{attribute 'GeneratedUsingTerminal: EL1262-0000-0002'}
{attribute addProperty BoxType "EL1262-0000-0002"}
{attribute addProperty Id "EtcSlaveTerminalBaseCh1_CycleCountAT %I*Ch1_CycleCount_9DBE2BC52Ch1_Input_0AT %I*Ch1_Input_FFC4CE241Ch1_Input_1AT %I*Ch1_Input_FFC4CE241Ch1_Input_2AT %I*Ch1_Input_FFC4CE241Ch1_Input_3AT %I*Ch1_Input_FFC4CE241Ch1_Input_4AT %I*Ch1_Input_FFC4CE241Ch1_Input_5AT %I*Ch1_Input_FFC4CE241Ch1_Input_6AT %I*Ch1_Input_FFC4CE241Ch1_Input_7AT %I*Ch1_Input_FFC4CE241Ch1_Input_8AT %I*Ch1_Input_FFC4CE241Ch1_Input_9AT %I*Ch1_Input_FFC4CE241GapAT %I*EMPTY_STRUCTURE0Ch2_CycleCountAT %I*Ch2_CycleCount_976A51B52Ch2_Input_0AT %I*Ch2_Input_78ADA90C1Ch2_Input_1AT %I*Ch2_Input_78ADA90C1Ch2_Input_2AT %I*Ch2_Input_78ADA90C1Ch2_Input_3AT %I*Ch2_Input_78ADA90C1Ch2_Input_4AT %I*Ch2_Input_78ADA90C1Ch2_Input_5AT %I*Ch2_Input_78ADA90C1Ch2_Input_6AT %I*Ch2_Input_78ADA90C1Ch2_Input_7AT %I*Ch2_Input_78ADA90C1Ch2_Input_8AT %I*Ch2_Input_78ADA90C1Ch2_Input_9AT %I*Ch2_Input_78ADA90C1Gap_1AT %I*EMPTY_STRUCTURE0NextSync1TimeAT %I*NextSync1Time_EE185E174WcStateAT %I*WcState_9091E0EB2InfoDataAT %I*InfoData_A7436BC610"}
{attribute addProperty CRC "3126613733"}
{attribute addProperty Size "40"}
TYPE EL1262_BA5C56E5 EXTENDS EtcSlaveTerminalBase :
STRUCT
	{attribute addProperty Name "Ch1_CycleCount"}
	Ch1_CycleCount : Ch1_CycleCount_9DBE2BC5;
	{attribute addProperty Name "Ch1_Input_0"}
	Ch1_Input_0 : Ch1_Input_FFC4CE24;
	{attribute addProperty Name "Ch1_Input_1"}
	Ch1_Input_1 : Ch1_Input_FFC4CE24;
	{attribute addProperty Name "Ch1_Input_2"}
	Ch1_Input_2 : Ch1_Input_FFC4CE24;
	{attribute addProperty Name "Ch1_Input_3"}
	Ch1_Input_3 : Ch1_Input_FFC4CE24;
	{attribute addProperty Name "Ch1_Input_4"}
	Ch1_Input_4 : Ch1_Input_FFC4CE24;
	{attribute addProperty Name "Ch1_Input_5"}
	Ch1_Input_5 : Ch1_Input_FFC4CE24;
	{attribute addProperty Name "Ch1_Input_6"}
	Ch1_Input_6 : Ch1_Input_FFC4CE24;
	{attribute addProperty Name "Ch1_Input_7"}
	Ch1_Input_7 : Ch1_Input_FFC4CE24;
	{attribute addProperty Name "Ch1_Input_8"}
	Ch1_Input_8 : Ch1_Input_FFC4CE24;
	{attribute addProperty Name "Ch1_Input_9"}
	Ch1_Input_9 : Ch1_Input_FFC4CE24;
	{attribute addProperty Name "Gap"}
	Gap : EMPTY_STRUCTURE;
	{attribute addProperty Name "Ch2_CycleCount"}
	Ch2_CycleCount : Ch2_CycleCount_976A51B5;
	{attribute addProperty Name "Ch2_Input_0"}
	Ch2_Input_0 : Ch2_Input_78ADA90C;
	{attribute addProperty Name "Ch2_Input_1"}
	Ch2_Input_1 : Ch2_Input_78ADA90C;
	{attribute addProperty Name "Ch2_Input_2"}
	Ch2_Input_2 : Ch2_Input_78ADA90C;
	{attribute addProperty Name "Ch2_Input_3"}
	Ch2_Input_3 : Ch2_Input_78ADA90C;
	{attribute addProperty Name "Ch2_Input_4"}
	Ch2_Input_4 : Ch2_Input_78ADA90C;
	{attribute addProperty Name "Ch2_Input_5"}
	Ch2_Input_5 : Ch2_Input_78ADA90C;
	{attribute addProperty Name "Ch2_Input_6"}
	Ch2_Input_6 : Ch2_Input_78ADA90C;
	{attribute addProperty Name "Ch2_Input_7"}
	Ch2_Input_7 : Ch2_Input_78ADA90C;
	{attribute addProperty Name "Ch2_Input_8"}
	Ch2_Input_8 : Ch2_Input_78ADA90C;
	{attribute addProperty Name "Ch2_Input_9"}
	Ch2_Input_9 : Ch2_Input_78ADA90C;
	{attribute addProperty Name "Gap_1"}
	Gap_1 : EMPTY_STRUCTURE;
	{attribute addProperty Name "NextSync1Time"}
	NextSync1Time : NextSync1Time_EE185E17;
	{attribute addProperty Name "WcState"}
	WcState : WcState_9091E0EB;
	{attribute addProperty Name "InfoData"}
	InfoData : InfoData_A7436BC6;
END_STRUCT
END_TYPE

(* stored: Version 1.2.0.0, ProductVersion 3.1.4024.9
   DUT EL1262_BA5C56E5: Id {edd9989f-dbf4-429e-84f6-4e01bcf50160} *)
